// TIA Portal V18 export
TYPE "LGasp_typeHMI_linea"
// stored: IsFailsafeCompliant false
   STRUCT
      NUMZONE : DInt;
      NUMDS : DInt;
      NUMSTAZIONI : DInt;
      NUMSAFETYDEVICE : DInt;
      NUMATTUATORI : DInt;
      NUMPUNZONATEARTICOLO : DInt;
      NUMRIGHEPRODUZIONE : DInt;
      NUMRIGHELISTATAGLI : DInt;
      NUMASSIAA : DInt;
      NUMPRGVALVOLE : DInt := 10;
      man : Bool;
      auto : Bool;
      semiauto { ExternalAccessible := 'False'; ExternalVisible := 'False'; ExternalWritable := 'False'} : Bool;
      MARCIAstop : Bool;
      allarmi : Bool;
      warning : Bool;
      nome_linea : WString[20];
      zona : Array[1.."N_ZONE"] of "LGasp_typeHMI_zona";
      stz : Array[1.."N_STAZIONI"] of "LGasp_typeHMI_stazione";
   END_STRUCT;
END_TYPE
